FUNCTION F_UpdateEventTimestampWithSystemTime
VAR_INPUT
	stEvent : Reference to ST_Event;
END_VAR
VAR
	fbGETSYSTEMTIME : GETSYSTEMTIME;
	
	stFileTime : T_FILETIME;
END_VAR

fbGETSYSTEMTIME(timeLoDW => stFileTime.dwLowDateTime,
				timeHiDW => stFileTIme.dwHighDateTime);
stEvent.dtTimestamp := FILETIME_TO_DT(fileTime := stFileTime);

END_FUNCTION

(* stored: Version 1.1.0.1, ProductVersion 3.1.4024.12
   POU F_UpdateEventTimestampWithSystemTime: Id {90d4bcb1-26f4-4eb7-bae3-1d2f76cf9b17}, SpecialFunc None *)
